{attribute 'GeneratedUsingTerminal: EL9550-0010-0016'}
{attribute addProperty BoxType "EL9550-0010-0016"}
{attribute addProperty Id "Status_UpAT %I*Status_Up_DB3531282Status_UsAT %I*Status_Us_DB3531282WcStateAT %I*WcState_9091E0EB2InfoDataAT %I*InfoData_6F19DB2B2"}
{attribute addProperty CRC "1048781225"}
{attribute addProperty Size "8"}
TYPE EL9550_3E8321A9 :
STRUCT
	{attribute addProperty Name "Status_Up"}
	Status_Up : Status_Up_DB353128;
	{attribute addProperty Name "Status_Us"}
	Status_Us : Status_Us_DB353128;
	{attribute addProperty Name "WcState"}
	WcState : WcState_9091E0EB;
	{attribute addProperty Name "InfoData"}
	InfoData : InfoData_6F19DB2B;
END_STRUCT
END_TYPE

(* stored: Version 1.2.0.0, ProductVersion 3.1.4024.9
   DUT EL9550_3E8321A9: Id {9405af90-7f56-483a-aa4e-342d48ce6889} *)
